// SIMATIC S7-200 SMART project (STEP 7-Micro/WIN SMART), CPU ST40

SYMBOL_TABLE 表格 1
                 T32      // 周期轮询时钟
                 T37      // 传送轮传感器延时
                 T38      // 传送轮传感器延时
                 T39      // 流程延时
                 T40      // 流程延时
                 T41      // 流程延时
                 VW1000   // 周期轮询计数器
                 VW2000   // 翻转速度
                 VW2500   // 升降速度
                 VD2010   // 翻转位置0
                 VD2020   // 翻转位置1  6881280
                 VD2510   // 升降位置最低 100
                 VD2520   // 升降位置中间  6000000
                 VD2530   // 升降位置最高  10850000
                 VD2540   // 升降位置存储
                 VD2550   // 升降位置1 3450000
                 VD2560   // 升降位置2 2000000
                 VW3000   // 翻转目标位置低八位
                 VW3002   // 翻转目标位置高八位
                 VW3100   // 翻转速度
                 VW3200   // 运行模式
                 VW3300   // 运行指令开始512
                 VW3400   // 运行指令清零0
                 VW3500   // 运行指令停止2
                 VW4000   // 升降目标位置低八位
                 VW4002   // 升降目标位置高八位
                 VW4100   // 升降速度
                 VD5000   // 升降实际位置
                 VD5100   // 升降中点与实际位置差值
                 VD5200   // 翻转实际位置
                 VD5300   // 翻转拿砖面与实际位置差值
                 VD5400   // 升降目标与实际位置差值
                 VD5500   // 翻转目标与实际位置差值
                 VW6000   // 检测是否到中点
                 VW6100   // 升降开始和结束标志位，0停止，1开始
                 VW6200   // 翻转开始和结束标志位，0停止，1开始
                 M21.0    // m21,0开始大循环控制
                 M5.0     // 传送轮
                 M20.0    // m20.0开始流程循环命令
END_SYMBOL_TABLE

SYMBOL_TABLE 系统符号
Always_On        SM0.0    // 始终接通
First_Scan_On    SM0.1    // 仅在第一个扫描周期时接通
END_SYMBOL_TABLE

ORGANIZATION_BLOCK MAIN:OB1
TITLE=程序注释
BEGIN
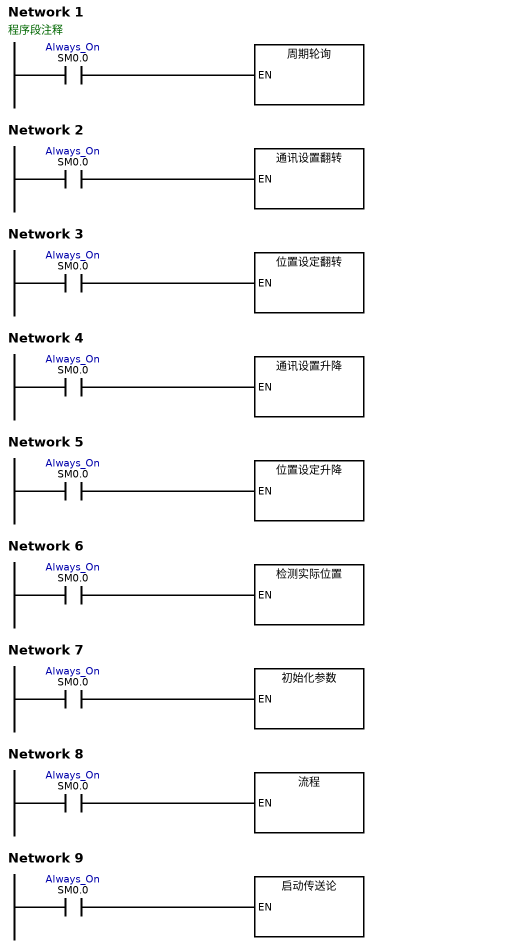
Network 1
// 程序段注释
LD     Always_On:SM0.0
CALL   周期轮询:SBR0
Network 2
LD     Always_On:SM0.0
CALL   通讯设置翻转:SBR1
Network 3
LD     Always_On:SM0.0
CALL   位置设定翻转:SBR5
Network 4
LD     Always_On:SM0.0
CALL   通讯设置升降:SBR6
Network 5
LD     Always_On:SM0.0
CALL   位置设定升降:SBR7
Network 6
LD     Always_On:SM0.0
CALL   检测实际位置:SBR8
Network 7
LD     Always_On:SM0.0
CALL   初始化参数:SBR9
Network 8
LD     Always_On:SM0.0
CALL   流程:SBR10
Network 9
LD     Always_On:SM0.0
CALL   启动传送论:SBR12
END_ORGANIZATION_BLOCK

SUBROUTINE_BLOCK 周期轮询:SBR0
TITLE=子程序注释
BEGIN
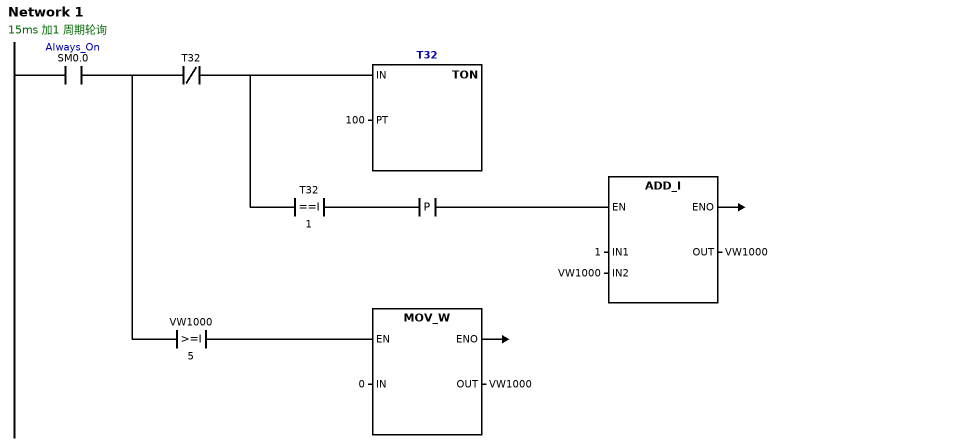
Network 1
// 15ms 加1 周期轮询
LD     Always_On:SM0.0
LPS
AN     T32
TON    T32, 100
AW=    T32, 1
EU
+I     1, VW1000
LPP
AW>=   VW1000, 5
MOVW   0, VW1000
END_SUBROUTINE_BLOCK

SUBROUTINE_BLOCK 通讯设置翻转:SBR1
TITLE=子程序注释
BEGIN
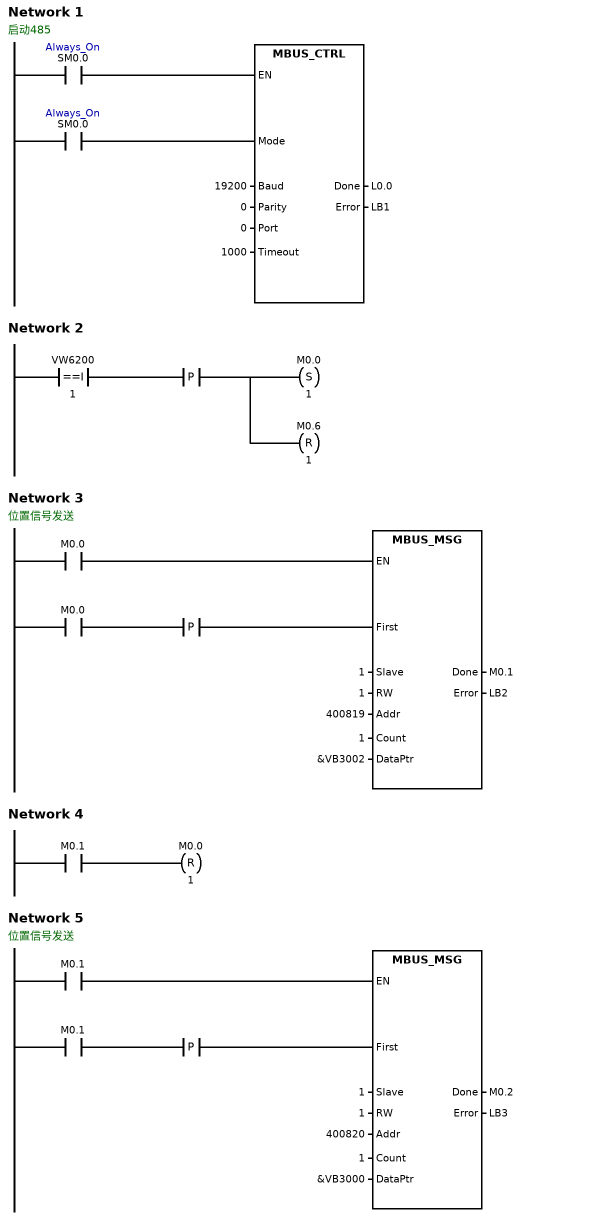
Network 1
// 启动485
LD     Always_On:SM0.0
=      L60.0
LD     Always_On:SM0.0
=      L63.7
LD     L60.0
CALL   MBUS_CTRL:SBR2, L63.7, 19200, 0, 0, 1000, L0.0, LB1
Network 2
LDW=   VW6200, 1
EU
S      M0.0, 1
R      M0.6, 1
Network 3
// 位置信号发送
LD     M0.0
=      L60.0
LD     M0.0
EU
=      L63.7
LD     L60.0
CALL   MBUS_MSG:SBR3, L63.7, 1, 1, 400819, 1, &VB3002, M0.1, LB2
Network 4
LD     M0.1
R      M0.0, 1
Network 5
// 位置信号发送
LD     M0.1
=      L60.0
LD     M0.1
EU
=      L63.7
LD     L60.0
CALL   MBUS_MSG:SBR3, L63.7, 1, 1, 400820, 1, &VB3000, M0.2, LB3
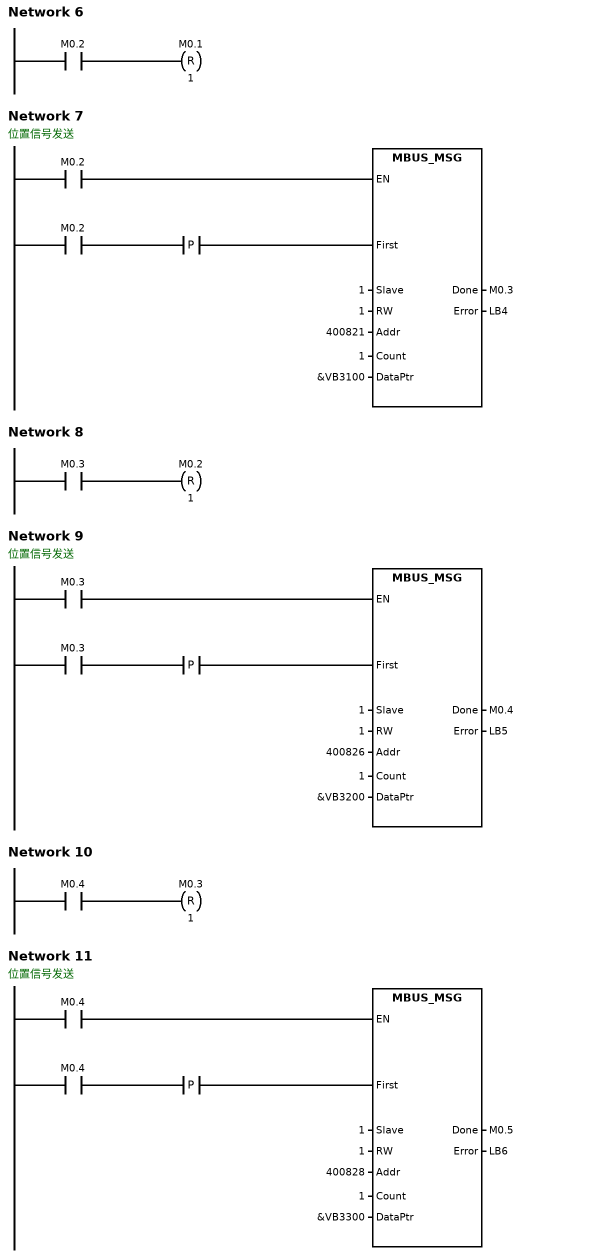
Network 6
LD     M0.2
R      M0.1, 1
Network 7
// 位置信号发送
LD     M0.2
=      L60.0
LD     M0.2
EU
=      L63.7
LD     L60.0
CALL   MBUS_MSG:SBR3, L63.7, 1, 1, 400821, 1, &VB3100, M0.3, LB4
Network 8
LD     M0.3
R      M0.2, 1
Network 9
// 位置信号发送
LD     M0.3
=      L60.0
LD     M0.3
EU
=      L63.7
LD     L60.0
CALL   MBUS_MSG:SBR3, L63.7, 1, 1, 400826, 1, &VB3200, M0.4, LB5
Network 10
LD     M0.4
R      M0.3, 1
Network 11
// 位置信号发送
LD     M0.4
=      L60.0
LD     M0.4
EU
=      L63.7
LD     L60.0
CALL   MBUS_MSG:SBR3, L63.7, 1, 1, 400828, 1, &VB3300, M0.5, LB6
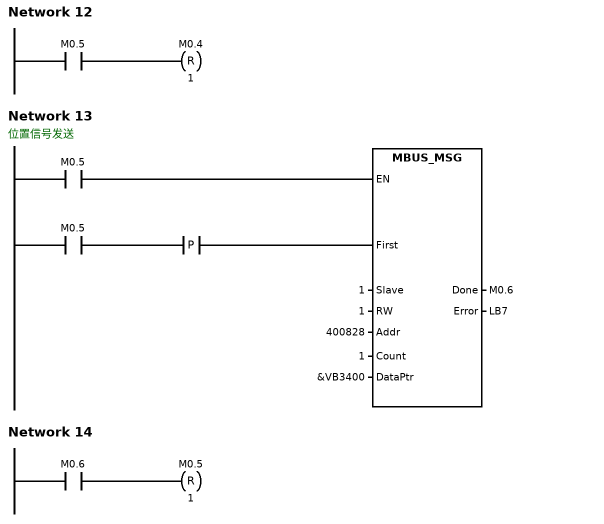
Network 12
LD     M0.5
R      M0.4, 1
Network 13
// 位置信号发送
LD     M0.5
=      L60.0
LD     M0.5
EU
=      L63.7
LD     L60.0
CALL   MBUS_MSG:SBR3, L63.7, 1, 1, 400828, 1, &VB3400, M0.6, LB7
Network 14
LD     M0.6
R      M0.5, 1
END_SUBROUTINE_BLOCK

// SBR2: protected block, not included

// SBR3: protected block, not included

// SBR4: protected block, not included

SUBROUTINE_BLOCK 位置设定翻转:SBR5
TITLE=子程序注释
BEGIN
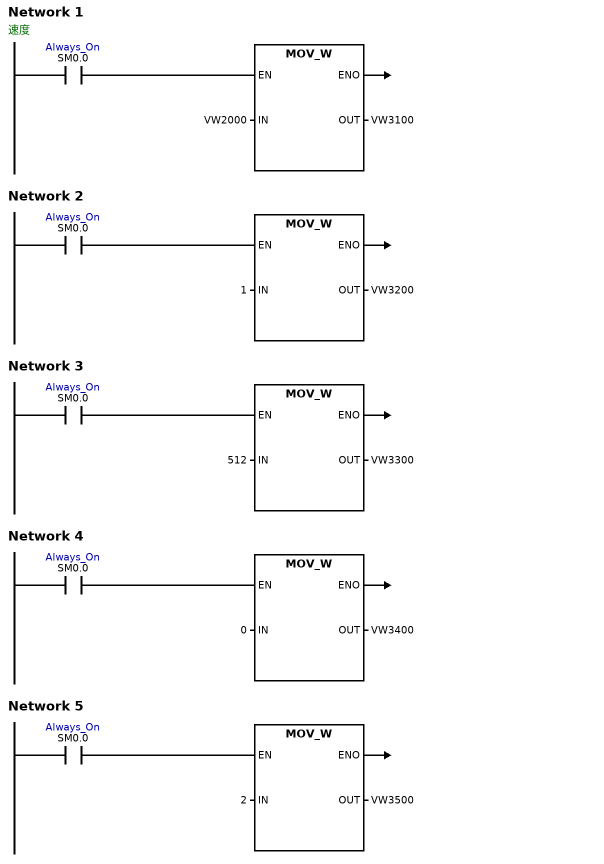
Network 1
// 速度
LD     Always_On:SM0.0
MOVW   VW2000, VW3100
Network 2
LD     Always_On:SM0.0
MOVW   1, VW3200
Network 3
LD     Always_On:SM0.0
MOVW   512, VW3300
Network 4
LD     Always_On:SM0.0
MOVW   0, VW3400
Network 5
LD     Always_On:SM0.0
MOVW   2, VW3500
END_SUBROUTINE_BLOCK

SUBROUTINE_BLOCK 通讯设置升降:SBR6
TITLE=子程序注释
BEGIN
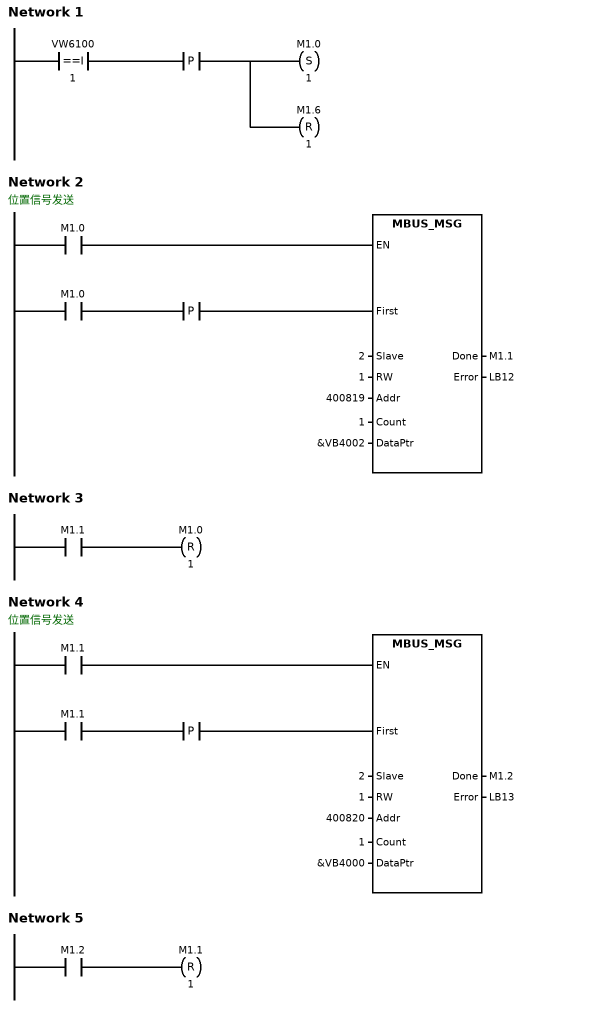
Network 1
LDW=   VW6100, 1
EU
S      M1.0, 1
R      M1.6, 1
Network 2
// 位置信号发送
LD     M1.0
=      L60.0
LD     M1.0
EU
=      L63.7
LD     L60.0
CALL   MBUS_MSG:SBR3, L63.7, 2, 1, 400819, 1, &VB4002, M1.1, LB12
Network 3
LD     M1.1
R      M1.0, 1
Network 4
// 位置信号发送
LD     M1.1
=      L60.0
LD     M1.1
EU
=      L63.7
LD     L60.0
CALL   MBUS_MSG:SBR3, L63.7, 2, 1, 400820, 1, &VB4000, M1.2, LB13
Network 5
LD     M1.2
R      M1.1, 1
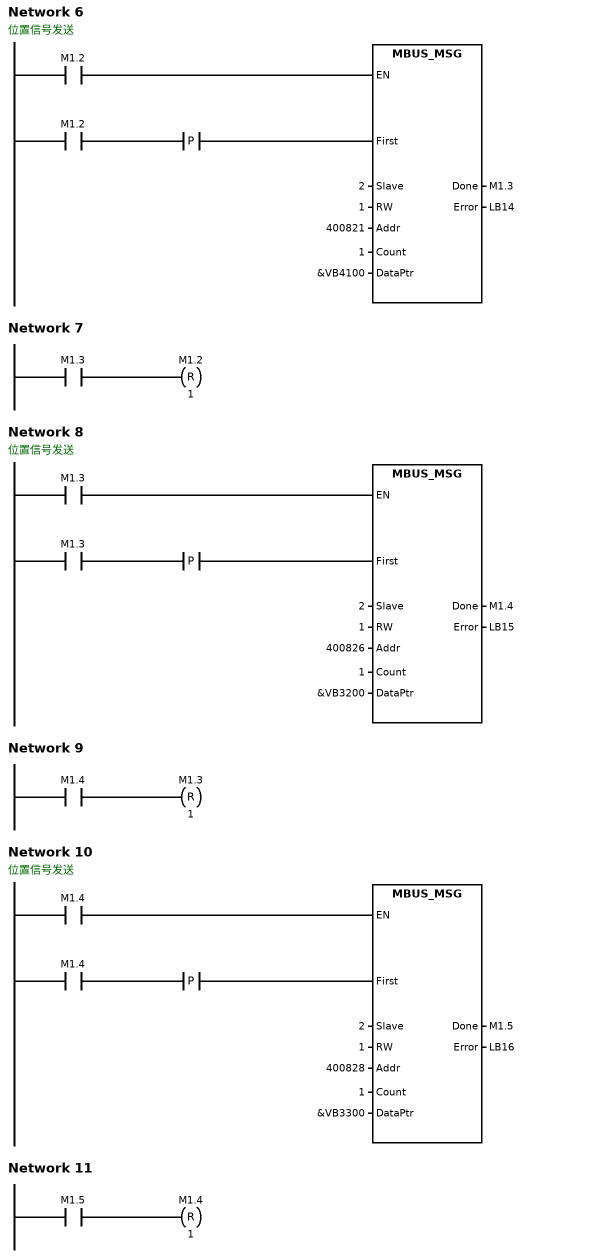
Network 6
// 位置信号发送
LD     M1.2
=      L60.0
LD     M1.2
EU
=      L63.7
LD     L60.0
CALL   MBUS_MSG:SBR3, L63.7, 2, 1, 400821, 1, &VB4100, M1.3, LB14
Network 7
LD     M1.3
R      M1.2, 1
Network 8
// 位置信号发送
LD     M1.3
=      L60.0
LD     M1.3
EU
=      L63.7
LD     L60.0
CALL   MBUS_MSG:SBR3, L63.7, 2, 1, 400826, 1, &VB3200, M1.4, LB15
Network 9
LD     M1.4
R      M1.3, 1
Network 10
// 位置信号发送
LD     M1.4
=      L60.0
LD     M1.4
EU
=      L63.7
LD     L60.0
CALL   MBUS_MSG:SBR3, L63.7, 2, 1, 400828, 1, &VB3300, M1.5, LB16
Network 11
LD     M1.5
R      M1.4, 1
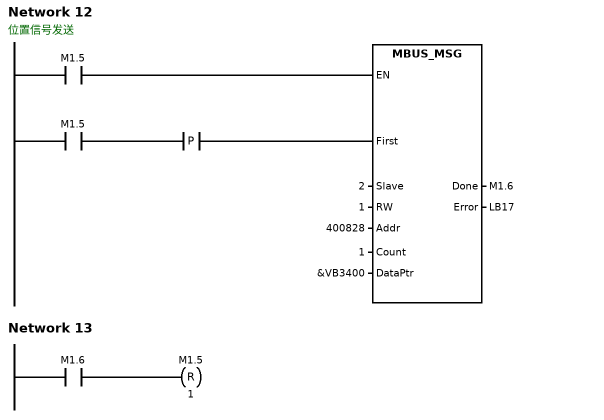
Network 12
// 位置信号发送
LD     M1.5
=      L60.0
LD     M1.5
EU
=      L63.7
LD     L60.0
CALL   MBUS_MSG:SBR3, L63.7, 2, 1, 400828, 1, &VB3400, M1.6, LB17
Network 13
LD     M1.6
R      M1.5, 1
Network 15
// 程序段注释
END_SUBROUTINE_BLOCK

SUBROUTINE_BLOCK 位置设定升降:SBR7
TITLE=子程序注释
BEGIN
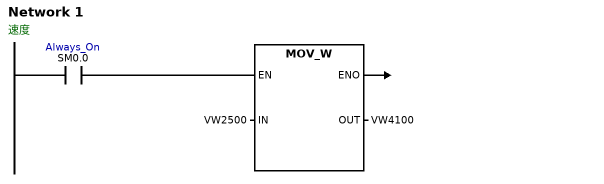
Network 1
// 速度
LD     Always_On:SM0.0
MOVW   VW2500, VW4100
END_SUBROUTINE_BLOCK

SUBROUTINE_BLOCK 检测实际位置:SBR8
TITLE=子程序注释
BEGIN
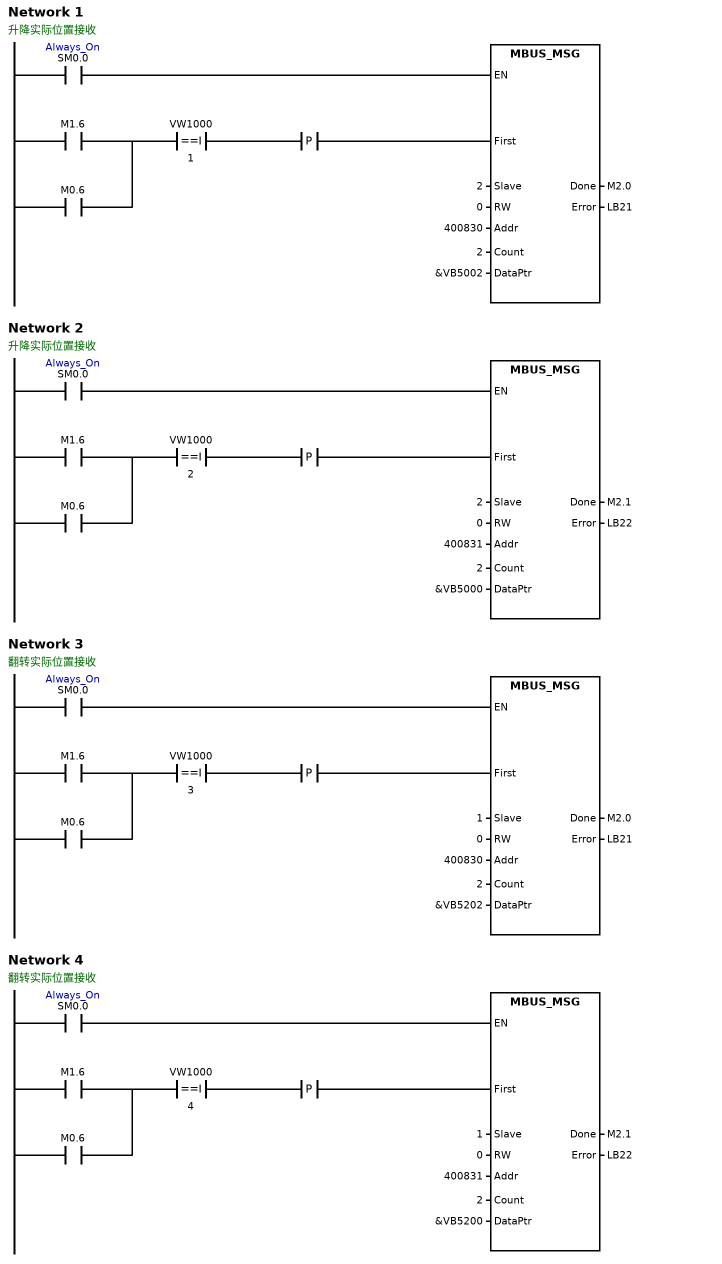
Network 1
// 升降实际位置接收
LD     Always_On:SM0.0
=      L60.0
LD     M1.6
O      M0.6
AW=    VW1000, 1
EU
=      L63.7
LD     L60.0
CALL   MBUS_MSG:SBR3, L63.7, 2, 0, 400830, 2, &VB5002, M2.0, LB21
Network 2
// 升降实际位置接收
LD     Always_On:SM0.0
=      L60.0
LD     M1.6
O      M0.6
AW=    VW1000, 2
EU
=      L63.7
LD     L60.0
CALL   MBUS_MSG:SBR3, L63.7, 2, 0, 400831, 2, &VB5000, M2.1, LB22
Network 3
// 翻转实际位置接收
LD     Always_On:SM0.0
=      L60.0
LD     M1.6
O      M0.6
AW=    VW1000, 3
EU
=      L63.7
LD     L60.0
CALL   MBUS_MSG:SBR3, L63.7, 1, 0, 400830, 2, &VB5202, M2.0, LB21
Network 4
// 翻转实际位置接收
LD     Always_On:SM0.0
=      L60.0
LD     M1.6
O      M0.6
AW=    VW1000, 4
EU
=      L63.7
LD     L60.0
CALL   MBUS_MSG:SBR3, L63.7, 1, 0, 400831, 2, &VB5200, M2.1, LB22
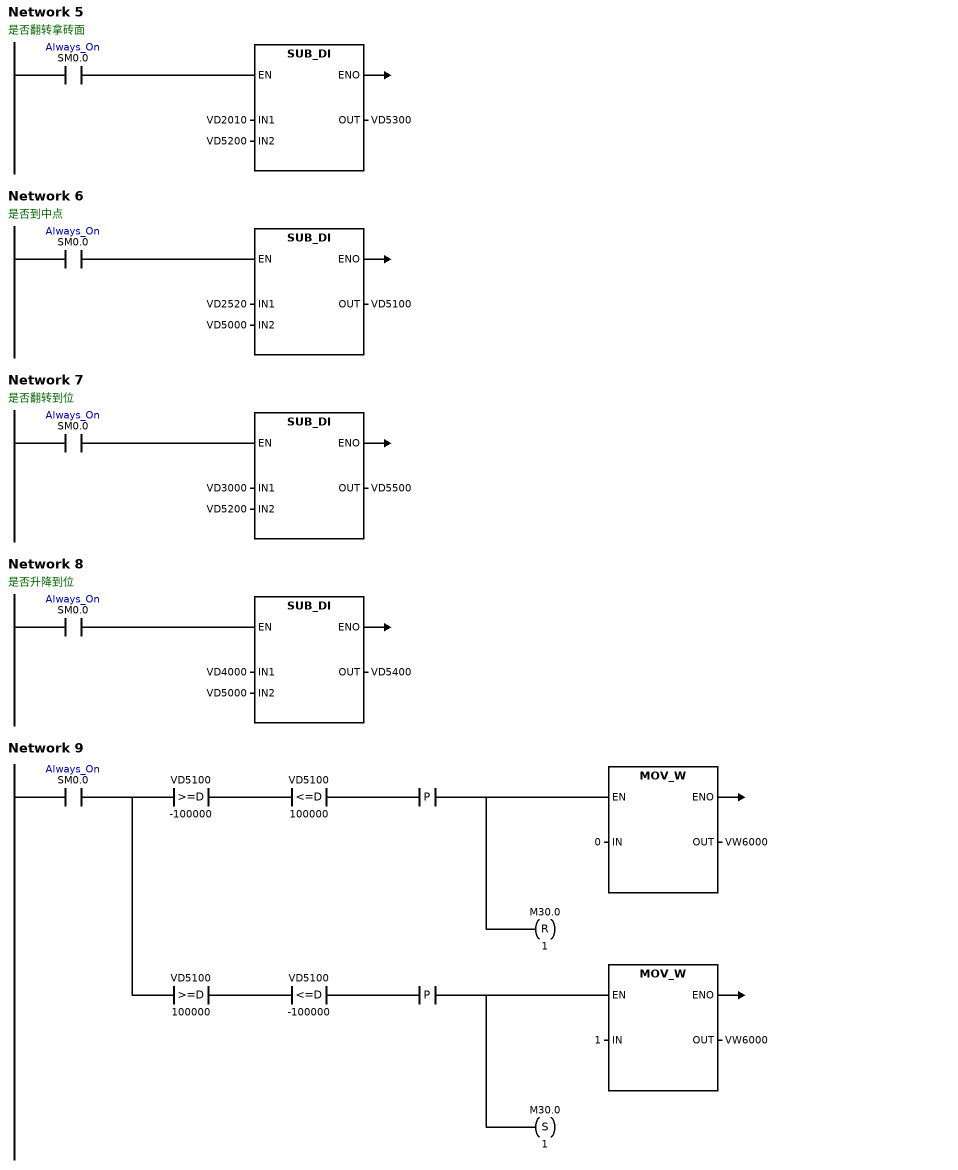
Network 5
// 是否翻转拿砖面
LD     Always_On:SM0.0
MOVD   VD2010, VD5300
-D     VD5200, VD5300
Network 6
// 是否到中点
LD     Always_On:SM0.0
MOVD   VD2520, VD5100
-D     VD5000, VD5100
Network 7
// 是否翻转到位
LD     Always_On:SM0.0
MOVD   VD3000, VD5500
-D     VD5200, VD5500
Network 8
// 是否升降到位
LD     Always_On:SM0.0
MOVD   VD4000, VD5400
-D     VD5000, VD5400
Network 9
LD     Always_On:SM0.0
LPS
AD>=   VD5100, -100000
AD<=   VD5100, 100000
EU
MOVW   0, VW6000
R      M30.0, 1
LPP
AD>=   VD5100, 100000
AD<=   VD5100, -100000
EU
MOVW   1, VW6000
S      M30.0, 1
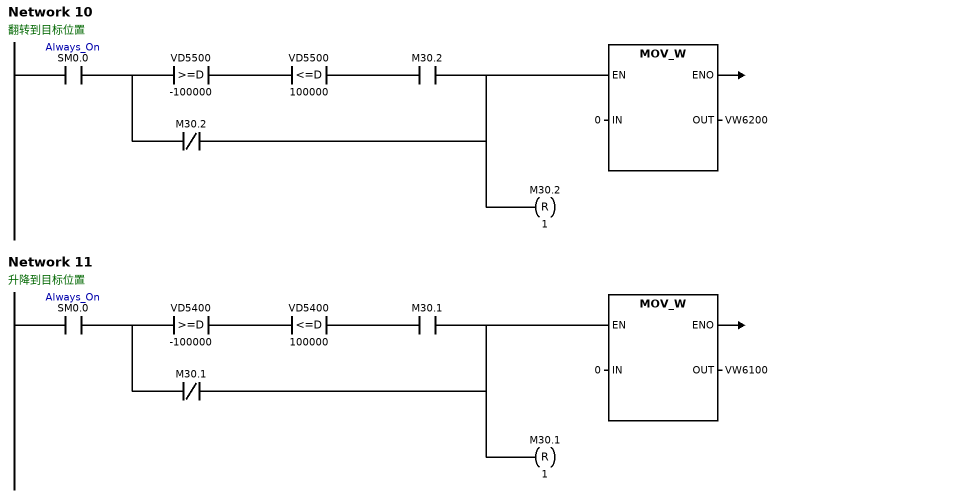
Network 10
// 翻转到目标位置
LD     Always_On:SM0.0
LDD>=  VD5500, -100000
AD<=   VD5500, 100000
A      M30.2
ON     M30.2
ALD
MOVW   0, VW6200
R      M30.2, 1
Network 11
// 升降到目标位置
LD     Always_On:SM0.0
LDD>=  VD5400, -100000
AD<=   VD5400, 100000
A      M30.1
ON     M30.1
ALD
MOVW   0, VW6100
R      M30.1, 1
END_SUBROUTINE_BLOCK

SUBROUTINE_BLOCK 初始化参数:SBR9
TITLE=子程序注释
BEGIN
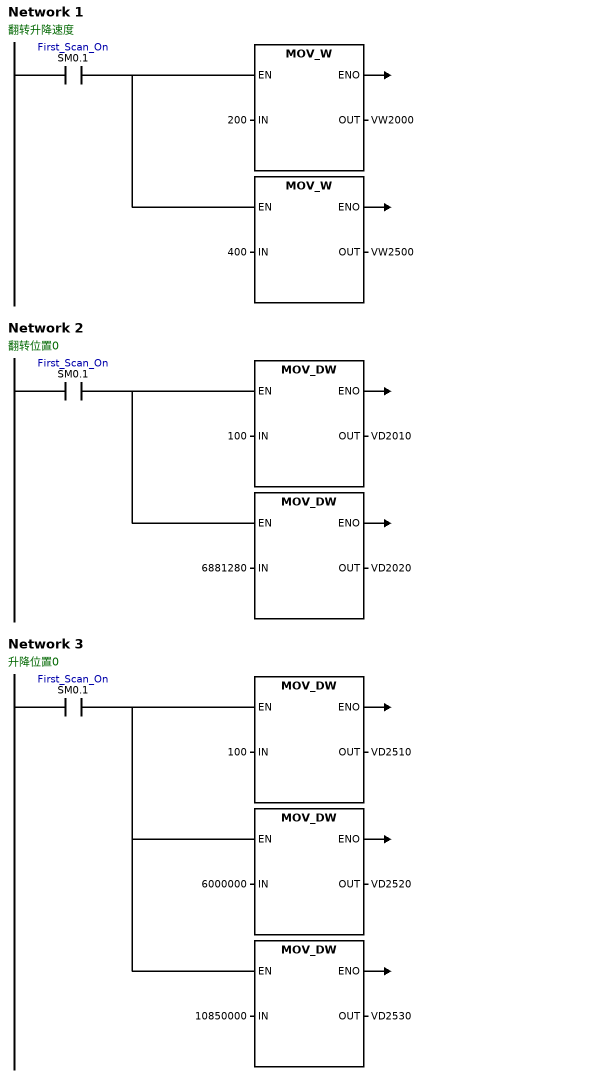
Network 1
// 翻转升降速度
LD     First_Scan_On:SM0.1
MOVW   200, VW2000
MOVW   400, VW2500
Network 2
// 翻转位置0
LD     First_Scan_On:SM0.1
MOVD   100, VD2010
MOVD   6881280, VD2020
Network 3
// 升降位置0
LD     First_Scan_On:SM0.1
MOVD   100, VD2510
MOVD   6000000, VD2520
MOVD   10850000, VD2530
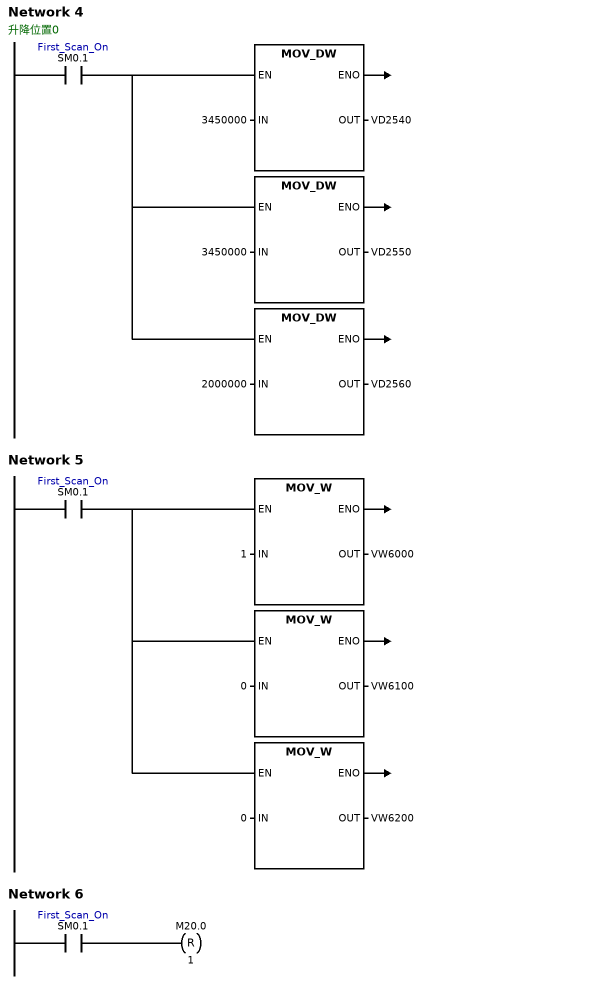
Network 4
// 升降位置0
LD     First_Scan_On:SM0.1
MOVD   3450000, VD2540
MOVD   3450000, VD2550
MOVD   2000000, VD2560
Network 5
LD     First_Scan_On:SM0.1
MOVW   1, VW6000
MOVW   0, VW6100
MOVW   0, VW6200
Network 6
LD     First_Scan_On:SM0.1
R      M20.0, 1
END_SUBROUTINE_BLOCK

SUBROUTINE_BLOCK 流程:SBR10
TITLE=
BEGIN
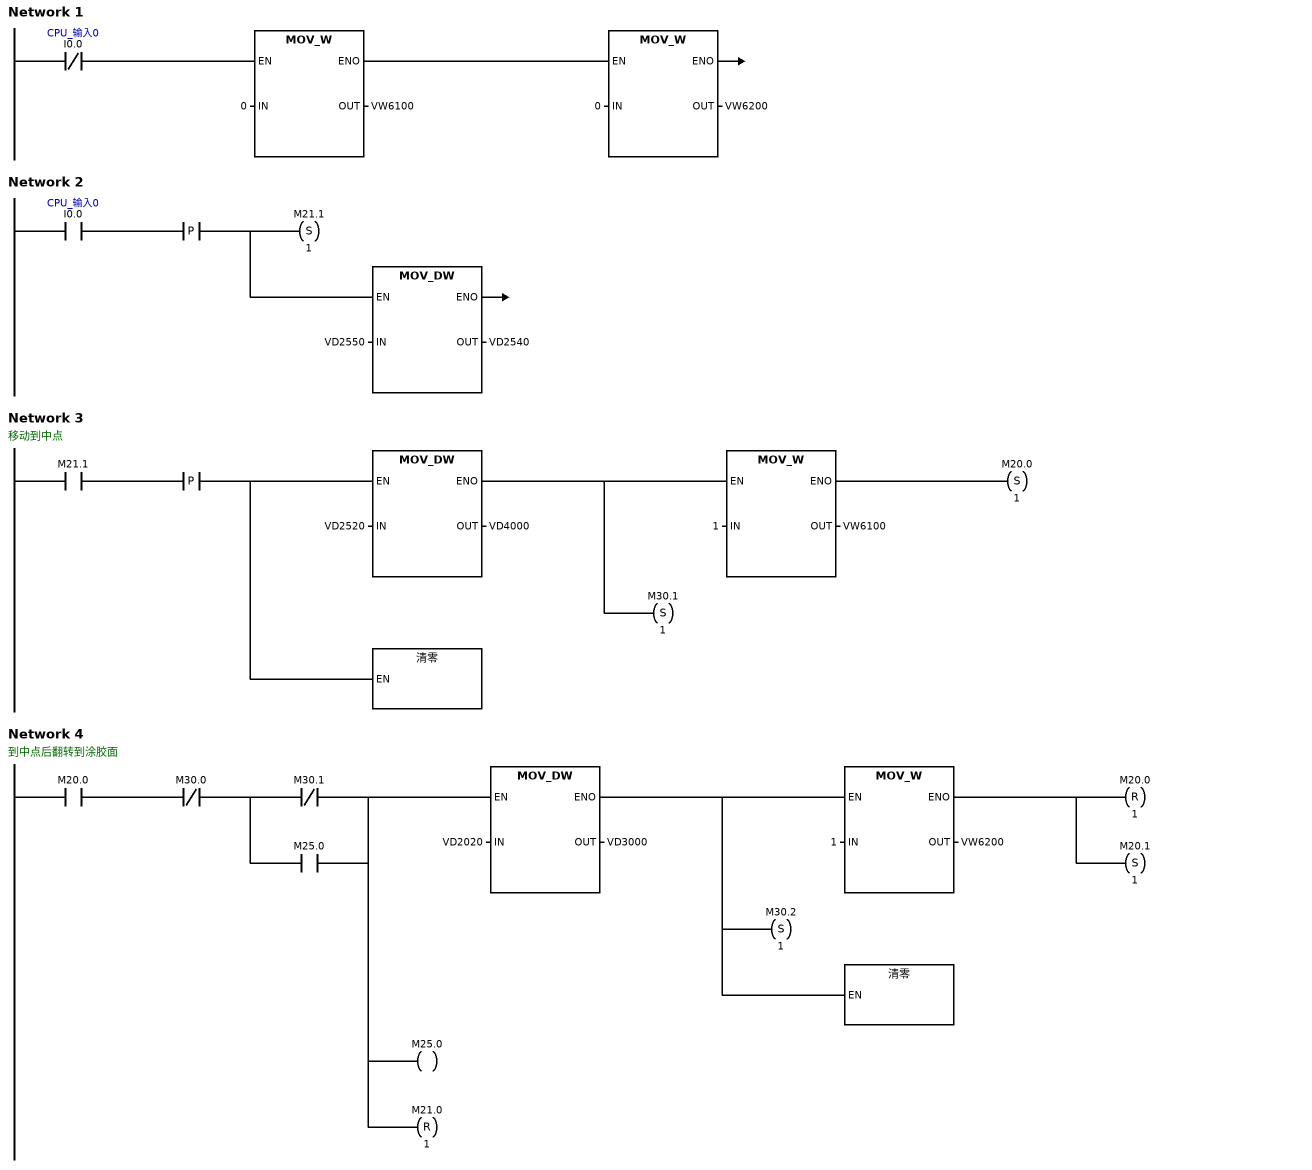
Network 1
LDN    CPU_输入0:I0.0
MOVW   0, VW6100
AENO
MOVW   0, VW6200
Network 2
LD     CPU_输入0:I0.0
EU
S      M21.1, 1
MOVD   VD2550, VD2540
Network 3
// 移动到中点
LD     M21.1
EU
LPS
MOVD   VD2520, VD4000
AENO
LPS
MOVW   1, VW6100
AENO
S      M20.0, 1
LPP
S      M30.1, 1
LPP
CALL   清零:SBR11
Network 4
// 到中点后翻转到涂胶面
LD     M20.0
AN     M30.0
LDN    M30.1
O      M25.0
ALD
LPS
MOVD   VD2020, VD3000
AENO
LPS
MOVW   1, VW6200
AENO
R      M20.0, 1
S      M20.1, 1
LPP
S      M30.2, 1
CALL   清零:SBR11
LPP
=      M25.0
R      M21.0, 1
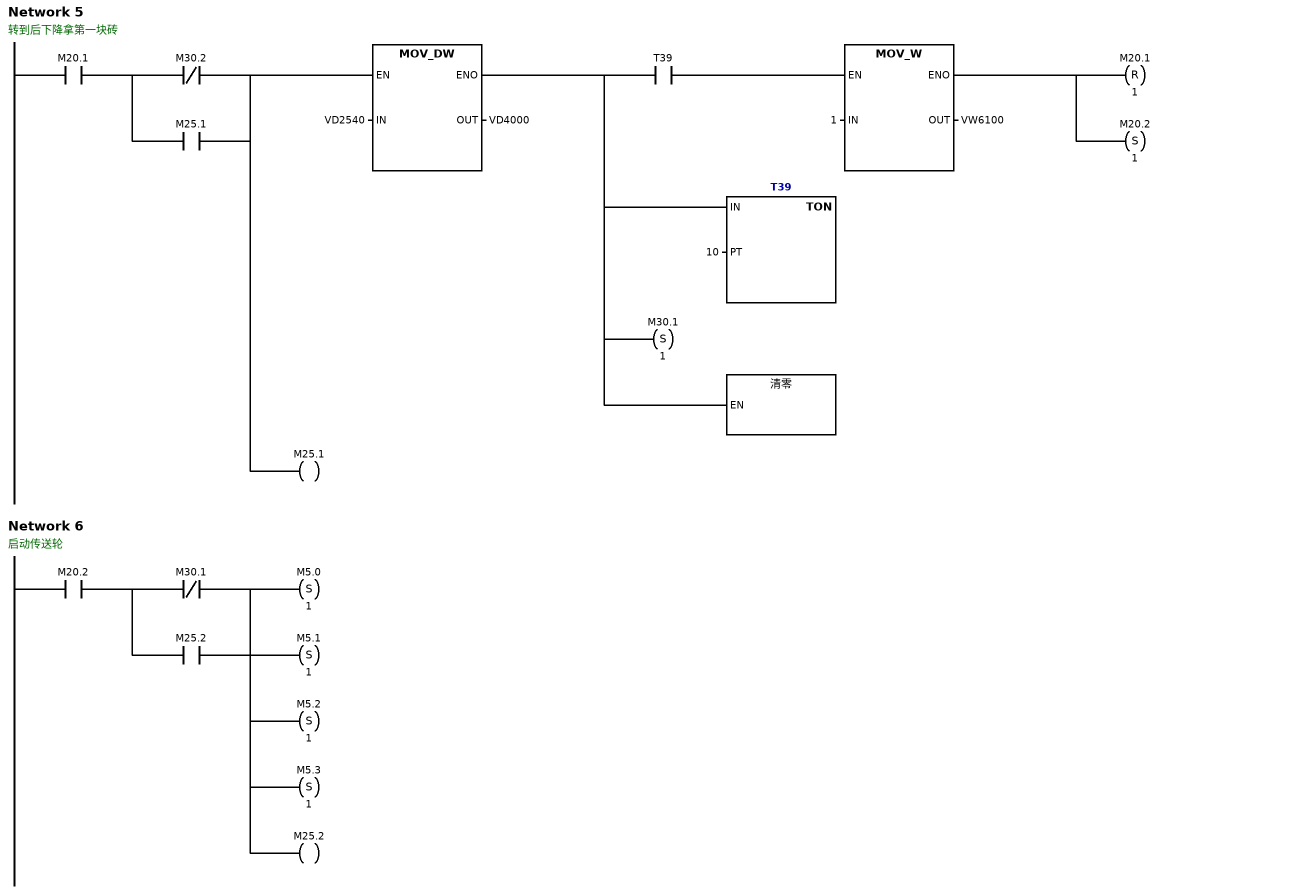
Network 5
// 转到后下降拿第一块砖
LD     M20.1
LDN    M30.2
O      M25.1
ALD
LPS
MOVD   VD2540, VD4000
AENO
LPS
A      T39
MOVW   1, VW6100
AENO
R      M20.1, 1
S      M20.2, 1
LPP
TON    T39, 10
S      M30.1, 1
CALL   清零:SBR11
LPP
=      M25.1
Network 6
// 启动传送轮
LD     M20.2
LDN    M30.1
O      M25.2
ALD
S      M5.0, 1
S      M5.1, 1
S      M5.2, 1
S      M5.3, 1
=      M25.2
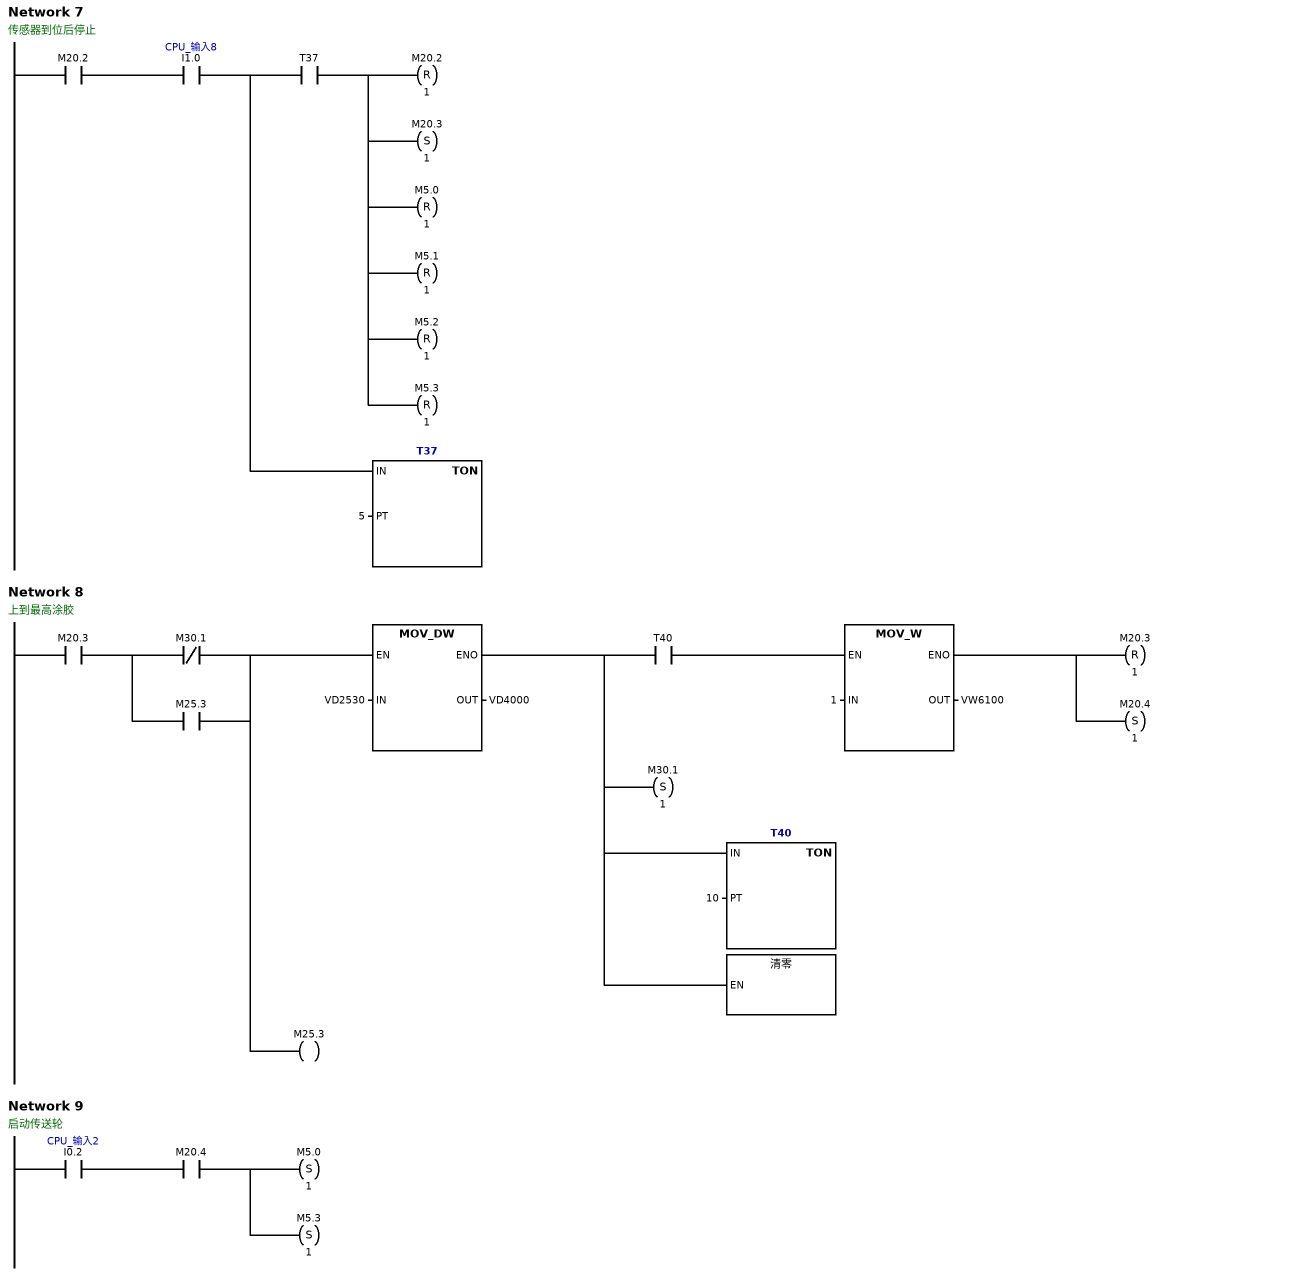
Network 7
// 传感器到位后停止
LD     M20.2
A      CPU_输入8:I1.0
LPS
A      T37
R      M20.2, 1
S      M20.3, 1
R      M5.0, 1
R      M5.1, 1
R      M5.2, 1
R      M5.3, 1
LPP
TON    T37, 5
Network 8
// 上到最高涂胶
LD     M20.3
LDN    M30.1
O      M25.3
ALD
LPS
MOVD   VD2530, VD4000
AENO
LPS
A      T40
MOVW   1, VW6100
AENO
R      M20.3, 1
S      M20.4, 1
LPP
S      M30.1, 1
TON    T40, 10
CALL   清零:SBR11
LPP
=      M25.3
Network 9
// 启动传送轮
LD     CPU_输入2:I0.2
A      M20.4
S      M5.0, 1
S      M5.3, 1
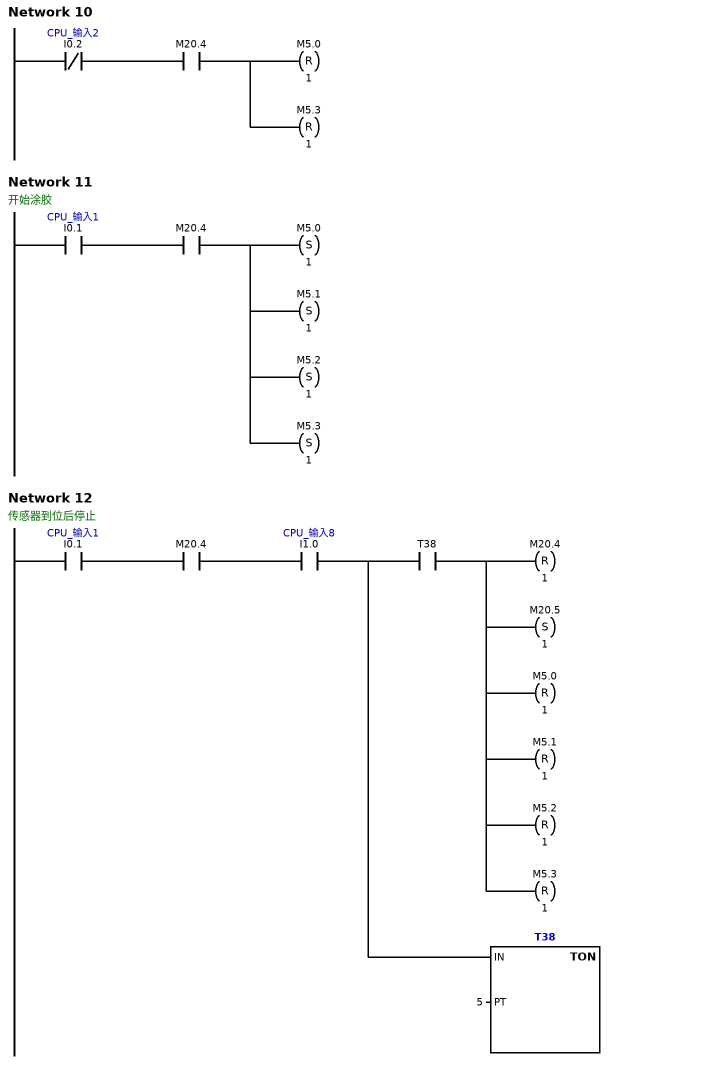
Network 10
LDN    CPU_输入2:I0.2
A      M20.4
R      M5.0, 1
R      M5.3, 1
Network 11
// 开始涂胶
LD     CPU_输入1:I0.1
A      M20.4
S      M5.0, 1
S      M5.1, 1
S      M5.2, 1
S      M5.3, 1
Network 12
// 传感器到位后停止
LD     CPU_输入1:I0.1
A      M20.4
A      CPU_输入8:I1.0
LPS
A      T38
R      M20.4, 1
S      M20.5, 1
R      M5.0, 1
R      M5.1, 1
R      M5.2, 1
R      M5.3, 1
LPP
TON    T38, 5
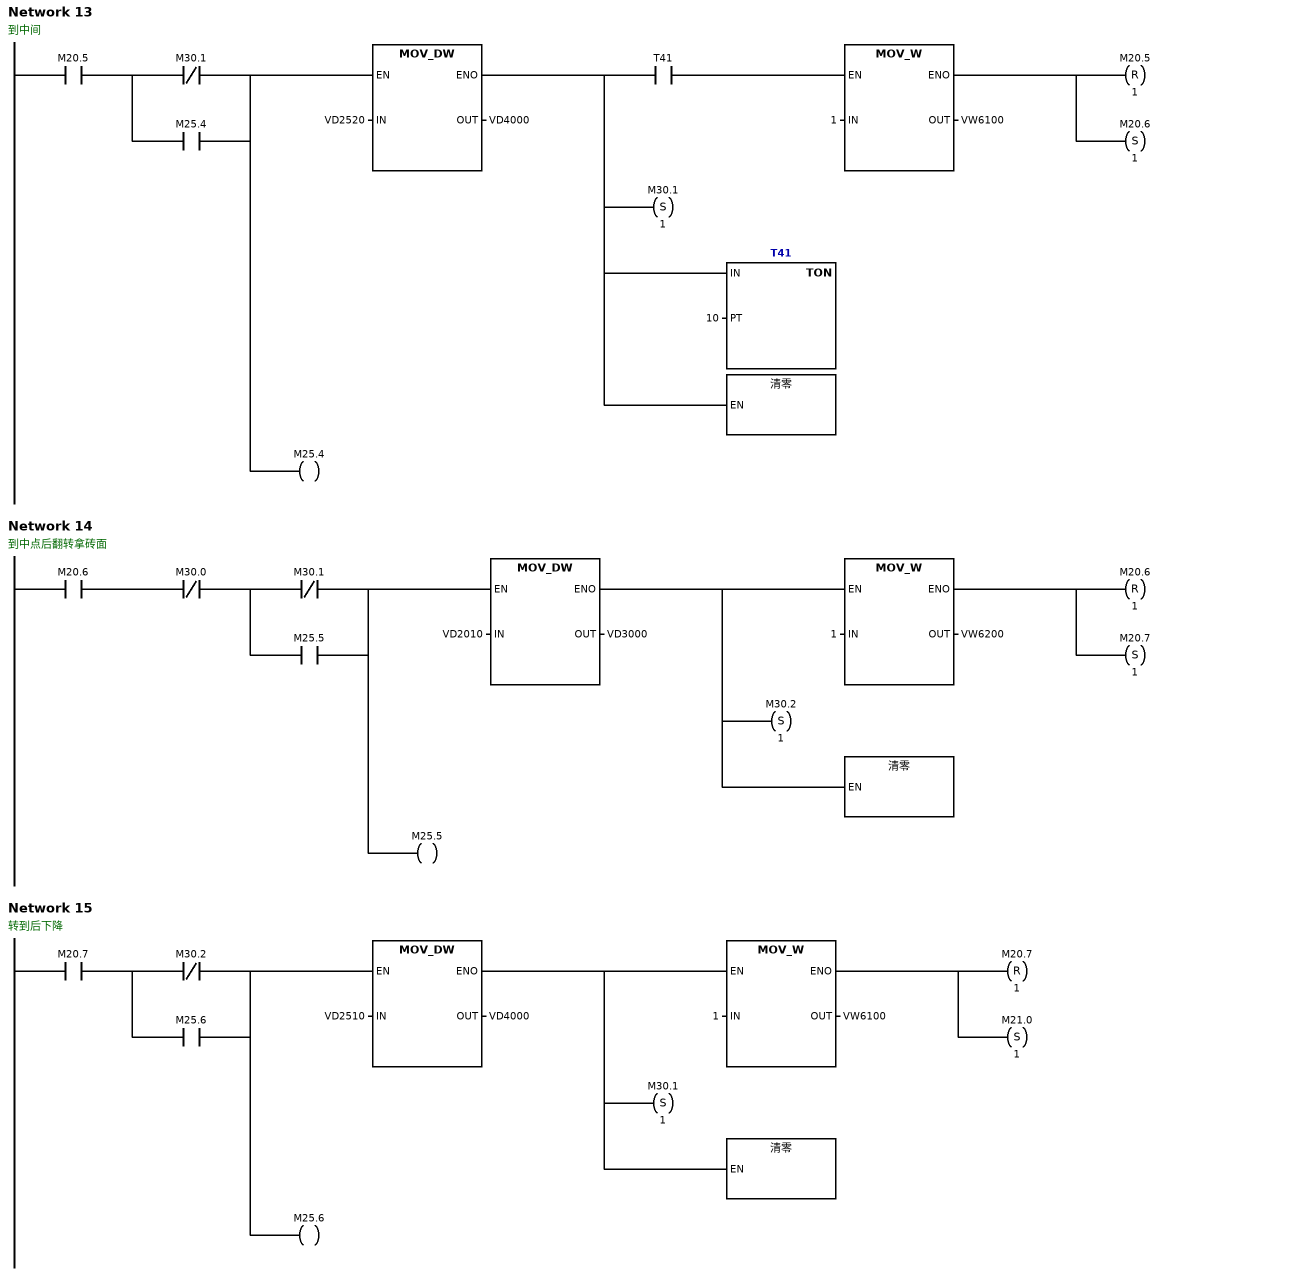
Network 13
// 到中间
LD     M20.5
LDN    M30.1
O      M25.4
ALD
LPS
MOVD   VD2520, VD4000
AENO
LPS
A      T41
MOVW   1, VW6100
AENO
R      M20.5, 1
S      M20.6, 1
LPP
S      M30.1, 1
TON    T41, 10
CALL   清零:SBR11
LPP
=      M25.4
Network 14
// 到中点后翻转拿砖面
LD     M20.6
AN     M30.0
LDN    M30.1
O      M25.5
ALD
LPS
MOVD   VD2010, VD3000
AENO
LPS
MOVW   1, VW6200
AENO
R      M20.6, 1
S      M20.7, 1
LPP
S      M30.2, 1
CALL   清零:SBR11
LPP
=      M25.5
Network 15
// 转到后下降
LD     M20.7
LDN    M30.2
O      M25.6
ALD
LPS
MOVD   VD2510, VD4000
AENO
LPS
MOVW   1, VW6100
AENO
R      M20.7, 1
S      M21.0, 1
LPP
S      M30.1, 1
CALL   清零:SBR11
LPP
=      M25.6
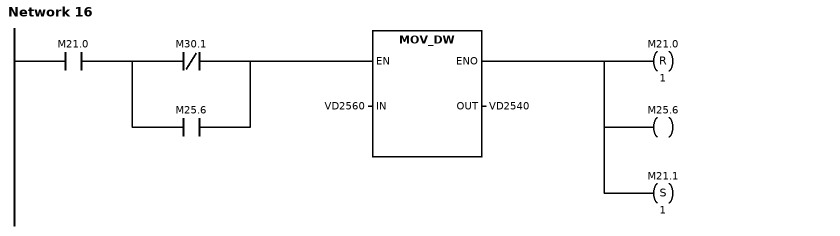
Network 16
LD     M21.0
LDN    M30.1
O      M25.6
ALD
MOVD   VD2560, VD2540
AENO
R      M21.0, 1
=      M25.6
S      M21.1, 1
END_SUBROUTINE_BLOCK

SUBROUTINE_BLOCK 清零:SBR11
TITLE=子程序注释
BEGIN
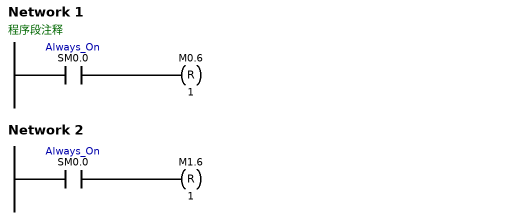
Network 1
// 程序段注释
LD     Always_On:SM0.0
R      M0.6, 1
Network 2
LD     Always_On:SM0.0
R      M1.6, 1
END_SUBROUTINE_BLOCK

SUBROUTINE_BLOCK 启动传送论:SBR12
TITLE=子程序注释
BEGIN
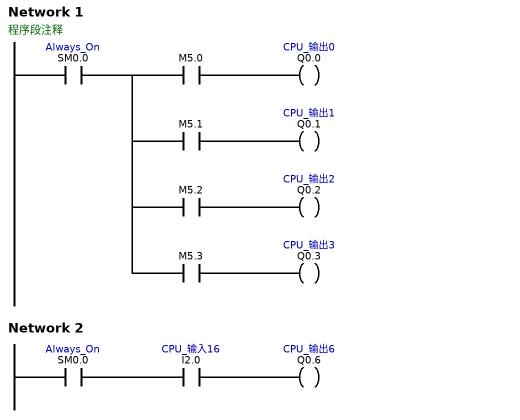
Network 1
// 程序段注释
LD     Always_On:SM0.0
LPS
A      M5.0
=      CPU_输出0:Q0.0
LRD
A      M5.1
=      CPU_输出1:Q0.1
LRD
A      M5.2
=      CPU_输出2:Q0.2
LPP
A      M5.3
=      CPU_输出3:Q0.3
Network 2
LD     Always_On:SM0.0
A      CPU_输入16:I2.0
=      CPU_输出6:Q0.6
END_SUBROUTINE_BLOCK
